FUNCTION_BLOCK PULSE_SOURCE (* IMpulse function source *)
  (* Standard: 61499-2 *)
  (* Version 11-01-12, GASR *)
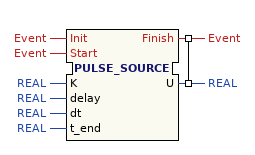
  EVENT_INPUT
    Init;
    Start;
  END_EVENT
  EVENT_OUTPUT
    Finish WITH U;
  END_EVENT
  VAR_INPUT
    K : REAL;
    delay : REAL;
    dt : REAL;
    t_end : REAL;
  END_VAR
  VAR_OUTPUT
    U : REAL;
  END_VAR
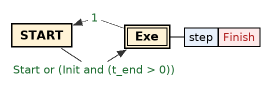
  EC_STATES
    Exe : step -> Finish;
    START;
  END_STATES
  EC_TRANSITIONS
    Exe TO START := 1;
    START TO Exe := Start or (Init and (t_end > 0));
  END_TRANSITIONS
  ALGORITHM step IN Lua:
if dt/2 >= delay and delay >= -dt/2 then  U = K end
t_end = t_end - dt
delay = delay - dt
  END_ALGORITHM
END_FUNCTION_BLOCK
